FUNCTION_BLOCK FB_DivertQueue EXTENDS RingBuffer.RingBufferMoverDivert
VAR
	nForCounterInterval			: UDINT;
	MoverDivert							: RingBuffer.ST_MoverDivert;
END_VAR

METHOD M_UpdateAtTrig
//Increment counter, mark each mover for divert interval
FOR nForCounterInterval := GC.nNumMinMovers TO GVL_General.nNumMovers DO
	
	IF (stSwitchStatus.ShuttleQueueCount + stSwitchStatus.ShuttleCountOnShortcut) <
		GVL_General.stSwitchConfig.SwitchModeInternal.MaxAllowedDivertCount THEN // command a mover to divert
			DivertQueue.P_MoverDivert.MoverID				:= DivertingMoverIndex;
			DivertQueue.P_MoverDivert.Divert				:= RingBuffer.E_Divert.Divert;
		IF (TempMoverIndex = GVL_General.stSwitchConfig.SwitchModeInternal.IntervalToDivert) THEN
			DivertQueue.P_MoverDivert.DivertOnInterval	:= TRUE;
		END_IF
			DivertQueue.AddObjToBuffer(RefObject := DivertQueue.P_MoverDivert);
			stSwitchStatus.ShuttleQueueCount := stSwitchStatus.ShuttleQueueCount + 1;
	END_IF

END_FOR
END_METHOD

PROPERTY P_MoverDivert : REFERENCE TO ST_MoverDivert
GET
P_MoverDivert REF= MoverDivert;
END_GET
END_PROPERTY

END_FUNCTION_BLOCK

(* stored: Version 1.1.0.1
   POU FB_DivertQueue: Id {6d05417c-3e76-051c-28a5-89303f3d9e18}, SpecialFunc None
   Method M_UpdateAtTrig: Id {6ebfa865-70ed-099f-252e-a28cbe294425}
   Property P_MoverDivert: Id {e439b90e-d481-0d68-25d8-af764ed57bd8}
   Get Get: Id {ac1dbd05-66a7-0918-1371-e3a68180d3c6} *)
